(* PLC project switch_2pos_1output, Dassault Systèmes ControlBuild 2024x *)
(* stored: creationDateTime 2023-10-03T11:13:22-01:00 *)

(* This module simulates a switch with 2 positions and 1 output. *)
FUNCTION_BLOCK equipment_library.switch_2pos_1output
  VAR_OUTPUT
    variable : BOOL := false;
  END_VAR
  VAR
    leftPosition : BOOL := false;
    rightPosition : BOOL := false;
  END_VAR

(* -----------------------------------------------------------------	*)
(* Type : Model of Operative Behaviour					*)
(* Category :  Power								*)
(* Author : Dassault Systemes						*)
(* Update date : June 2018							*)
(* -----------------------------------------------------------------	*)
(* This module simulates a switch with 2 positions and 1 output.	*)
(* -----------------------------------------------------------------	*)


IF (leftPosition) THEN
	variable := FALSE;
END_IF;
IF (rightPosition) THEN
	variable := TRUE;
END_IF;
leftPosition := FALSE;
rightPosition := FALSE;
END_FUNCTION_BLOCK
